// TIA Portal V17 export
// export: Created 2023-12-22T15:05:35.4887265Z, ExportSetting WithDefaults, DisplayName Totally Integrated Automation Portal, DisplayVersion V17, DisplayName TIA Portal Openness, DisplayVersion V17, DisplayName TIA Portal Version Control Interface, DisplayVersion V17, DisplayName STEP 7 Professional, DisplayVersion V17, DisplayName STEP 7 Safety, DisplayVersion V17, DisplayName WinCC Advanced, DisplayVersion V17
TYPE "Out_AI"
// stored: IsFailsafeCompliant false
   STRUCT
      Result : Real;   // Показания датчика
      Converter : Struct   // Масштабирование сигнала
         Min_Out { S7_SetPoint := 'True'} : Real;   // Минимальный выходной сигнал
         Max_Out { S7_SetPoint := 'True'} : Real := 100.0;   // Максимальный выходной сигнал
      END_STRUCT;
      Alarms : Word;   // Слово аварий
      SP : Struct   // Уставки аварий
         HH { S7_SetPoint := 'True'} : Real := 90.0;
         H { S7_SetPoint := 'True'} : Real := 85.0;
         L { S7_SetPoint := 'True'} : Real := 15.0;
         LL { S7_SetPoint := 'True'} : Real := 10.0;
      END_STRUCT;
   END_STRUCT;
END_TYPE
